FUNCTION_BLOCK MockObject EXTENDS Object
VAR
	_isRegistered : BOOL;
END_VAR

METHOD IsRegistered : BOOL
VAR_INPUT
END_VAR
IsRegistered := _isRegistered;
END_METHOD

METHOD RegisterWithParent
VAR_INPUT
	Parent	: I_HostObjects;
END_VAR
IF NOT _isRegistered THEN
	IF SUCCEEDED(Parent.RegisterObject(THIS^)) THEN
		_isRegistered := TRUE;
	ELSE
		_isRegistered := FALSE;
	END_IF
END_IF
END_METHOD

END_FUNCTION_BLOCK

(* stored: Version 1.1.0.1
   POU MockObject: Id {6f8b0af1-76ba-4e84-8c37-25fa8b1ced80}, SpecialFunc None
   Method IsRegistered: Id {cffa730f-5549-42cb-a928-e7485adf8a67}
   Method RegisterWithParent: Id {7e21115c-4d61-41fa-a740-8dd9357bf43a} *)
